// Bandrundlauf-Controller
// Kontrolliert den Bandrundlauf, ist eigentlich der Hauptbaustein(deshalb wird direkt auf PLC-Variablen zugegriffen(ohne Schnittstellenübergabe)
FUNCTION_BLOCK FB_ConvSys
VAR
    vsFB_ConvPurple : FB_Conveyor;
    vsFB_ConvOrange : FB_Conveyor;
    vsFB_ConvYellow : FB_Conveyor;
    vsFB_ConvBlue : FB_Conveyor;

    vsFB_CounterR : CTU := (PV := 0);
	vsFB_CounterL : FB_MyUpCounter;

    // Enumeration for state machine, conveyor
    eStateConveyor : E_StateConveyor;

    fbChrono : FB_Chrono;
    fbConvLapTimeStatistic : FB_ConvStatistic;
	// Maximale Rundenzeit der 10 letzten Umläufe
	tMaxLapTime: TIME;
END_VAR

// Conveyor state machine
CASE eStateConveyor OF
    E_StateConveyor.C_INIT:
        GVL_SimitSp.Qx_MotorAcwPurple := FALSE;
        GVL_SimitSp.Qx_MotorCwPurple := FALSE;
        GVL_SimitSp.Qx_FullSpeedPurple := FALSE;
        GVL_SimitSp.Qx_MotorAcwOrange := FALSE;
        GVL_SimitSp.Qx_MotorCwOrange := FALSE;
        GVL_SimitSp.Qx_FullSpeedOrange := FALSE;
        GVL_SimitSp.Qx_MotorAcwYellow := FALSE;
        GVL_SimitSp.Qx_MotorCwYellow := FALSE;
        GVL_SimitSp.Qx_FullSpeedYellow := FALSE;
        GVL_SimitSp.Qx_MotorAcwBlue := FALSE;
        GVL_SimitSp.Qx_MotorCwBlue := FALSE;
        GVL_SimitSp.Qx_FullSpeedBlue := FALSE;
        eStateConveyor := E_StateConveyor.C_NORMAL;

    E_StateConveyor.C_NORMAL:
        vsFB_ConvPurple.vix_Left := GVL_SimitSp.Ix_Left;
        vsFB_ConvPurple.vix_Right := GVL_SimitSp.Ix_Right;
        vsFB_ConvOrange.vix_Left := GVL_SimitSp.Ix_Left;
        vsFB_ConvOrange.vix_Right := GVL_SimitSp.Ix_Right;
        vsFB_ConvYellow.vix_Left := GVL_SimitSp.Ix_Left;
        vsFB_ConvYellow.vix_Right := GVL_SimitSp.Ix_Right;
        vsFB_ConvBlue.vix_Left := GVL_SimitSp.Ix_Left;
        vsFB_ConvBlue.vix_Right := GVL_SimitSp.Ix_Right;

        IF GVL_SimitSp.Ix_Enable THEN
            GVL_SimitSp.Qx_LightGreen := TRUE;
            eStateConveyor := E_StateConveyor.C_INIT_PROCESS;
        END_IF

    E_StateConveyor.C_INIT_PROCESS:
        vsFB_ConvPurple.vix_Left := FALSE;
        vsFB_ConvPurple.vix_Right := TRUE;
        vsFB_ConvOrange.vix_Left := FALSE;
        vsFB_ConvOrange.vix_Right := TRUE;
        vsFB_ConvYellow.vix_Left := FALSE;
        vsFB_ConvYellow.vix_Right := TRUE;
        vsFB_ConvBlue.vix_Left := FALSE;
        vsFB_ConvBlue.vix_Right := TRUE;

        eStateConveyor := E_StateConveyor.C_PURPLE_BACK;

    E_StateConveyor.C_PURPLE_BACK:
        IF GVL_SimitSp.Ix_RSensorPurple THEN
            vsFB_ConvPurple.vix_Left := TRUE;
            vsFB_ConvPurple.vix_Right := FALSE;

            eStateConveyor := E_StateConveyor.C_PURPLE_FORWARD;
        END_IF

    E_StateConveyor.C_PURPLE_FORWARD:
        IF GVL_SimitSp.Ix_LSensorPurple THEN
            vsFB_ConvPurple.vix_Left := FALSE;
            vsFB_ConvPurple.vix_Right := TRUE;

            eStateConveyor := E_StateConveyor.C_ORANGE_BACK;
        END_IF

    E_StateConveyor.C_ORANGE_BACK:
        IF GVL_SimitSp.Ix_RSensorOrange THEN
            vsFB_ConvOrange.vix_Left := TRUE;
            vsFB_ConvOrange.vix_Right := FALSE;

            eStateConveyor := E_StateConveyor.C_ORANGE_FORWARD;
        END_IF

    E_StateConveyor.C_ORANGE_FORWARD:
        IF GVL_SimitSp.Ix_LSensorOrange THEN
            vsFB_Convorange.vix_Left := FALSE;
            vsFB_Convorange.vix_Right := TRUE;

            eStateConveyor := E_StateConveyor.C_YELLOW_BACK;
        END_IF

    E_StateConveyor.C_YELLOW_BACK:
        IF GVL_SimitSp.Ix_RSensorYellow THEN
            vsFB_ConvYellow.vix_Left := TRUE;
            vsFB_ConvYellow.vix_Right := FALSE;

            eStateConveyor := E_StateConveyor.C_YELLOW_FORWARD;
        END_IF

    E_StateConveyor.C_YELLOW_FORWARD:
        IF GVL_SimitSp.Ix_LSensorYellow THEN
            vsFB_Convyellow.vix_Left := FALSE;
            vsFB_Convyellow.vix_Right := TRUE;

            eStateConveyor := E_StateConveyor.C_BLUE_BACK;
        END_IF

    E_StateConveyor.C_BLUE_BACK:
        IF GVL_SimitSp.Ix_RSensorBlue THEN
            vsFB_ConvBlue.vix_Left := TRUE;
            vsFB_ConvBlue.vix_Right := FALSE;

            eStateConveyor := E_StateConveyor.C_BLUE_FORWARD;
        END_IF

    E_StateConveyor.C_BLUE_FORWARD:
        IF GVL_SimitSp.Ix_LSensorblue THEN
            vsFB_Convblue.vix_Left := FALSE;
            vsFB_Convblue.vix_Right := TRUE;

            eStateConveyor := E_StateConveyor.C_PURPLE_BACK;
        END_IF

    ELSE
        eStateConveyor := E_StateConveyor.C_INIT;
END_CASE

// Reset conveyor state machine
IF GVL_SimitSp.Ix_Reset THEN
    eStateConveyor := E_StateConveyor.C_INIT;
END_IF

(*Multiinstanzaufruf von Band lila*)
vsFB_ConvPurple(vix_Power := GVL_SimitSp.Ix_PowerOn,
                vix_On := GVL_SimitSp.Ix_On,
                vix_Off := GVL_SimitSp.Ix_Off,
                vix_ManAuto := GVL_SimitSp.Ix_ManAuto,
                viw_Speed := GVL_SimitSp.Iw_SliderValue,
                vqx_MotorCw => GVL_SimitSp.Qx_MotorCwPurple,
                vqx_MotorAcw => GVL_SimitSp.Qx_MotorAcwPurple,
                vqx_VarSpeed => GVL_SimitSp.Qx_EnableVarSpeedPurple,
                vqw_Speed => GVL_SimitSp.Qw_VarSpeedPurple);
     
(*Multiinstanzaufruf von Band orange*)
vsFB_ConvOrange(vix_Power := GVL_SimitSp.Ix_PowerOn,
                vix_On := GVL_SimitSp.Ix_On,
                vix_Off := GVL_SimitSp.Ix_Off,
                vix_ManAuto := GVL_SimitSp.Ix_ManAuto,
                viw_Speed := GVL_SimitSp.Iw_SliderValue,
                vqx_MotorCw => GVL_SimitSp.Qx_MotorCwOrange,
                vqx_MotorAcw => GVL_SimitSp.Qx_MotorAcwOrange,
                vqx_VarSpeed => GVL_SimitSp.Qx_EnableVarSpeedOrange,
                vqw_Speed => GVL_SimitSp.Qw_VarSpeedOrange);

(*Multiinstanzaufruf von Band yellow*)
vsFB_ConvYellow(vix_Power := GVL_SimitSp.Ix_PowerOn,
                vix_On := GVL_SimitSp.Ix_On,
                vix_Off := GVL_SimitSp.Ix_Off,
                vix_ManAuto := GVL_SimitSp.Ix_ManAuto,
                viw_Speed := GVL_SimitSp.Iw_SliderValue,
                vqx_MotorCw => GVL_SimitSp.Qx_MotorCwYellow,
                vqx_MotorAcw => GVL_SimitSp.Qx_MotorAcwYellow,
                vqx_VarSpeed => GVL_SimitSp.Qx_EnableVarSpeedYellow,
                vqw_Speed => GVL_SimitSp.Qw_VarSpeedYellow);

(*Multiinstanzaufruf von Band blue*)
vsFB_ConvBlue(vix_Power := GVL_SimitSp.Ix_PowerOn,
                vix_On := GVL_SimitSp.Ix_On,
                vix_Off := GVL_SimitSp.Ix_Off,
                vix_ManAuto := GVL_SimitSp.Ix_ManAuto,
                viw_Speed := GVL_SimitSp.Iw_SliderValue,
                vqx_MotorCw => GVL_SimitSp.Qx_MotorCwBlue,
                vqx_MotorAcw => GVL_SimitSp.Qx_MotorAcwBlue,
                vqx_VarSpeed => GVL_SimitSp.Qx_EnableVarSpeedBlue,
                vqw_Speed => GVL_SimitSp.Qw_VarSpeedBlue);

(*Rundlauf Anzeigen*)
GVL_SimitSp.Qx_LightBlue := GVL_SimitSp.Qx_MotorAcwBlue;  (*Gegenuhrzeigersinn Kontrolleuchte*)
GVL_SimitSp.Qx_LightYellow := GVL_SimitSp.Qx_MotorCwBlue; (*Uhrzeigersinn Kontrolleuchte*)
GVL_SimitSp.Qw_Display := GVL_SimitSp.Qw_VarSpeedPurple;  (*aktuelle variable Geschwindigkeit*)

(*Eilgang auf Enable Taster*)
GVL_SimitSp.Qx_FullSpeedPurple := GVL_SimitSp.Ix_Enable;
GVL_SimitSp.Qx_FullSpeedOrange := GVL_SimitSp.Ix_Enable;
GVL_SimitSp.Qx_FullSpeedYellow := GVL_SimitSp.Ix_Enable;
GVL_SimitSp.Qx_FullSpeedBlue := GVL_SimitSp.Ix_Enable; 

// Conveyor circulation counter right
vsFB_CounterR(CU := GVL_SimitSp.Ix_RSensorPurple AND GVL_SimitSp.Qx_MotorAcwPurple);
GVL_SimitSp.Qb_74 := WORD_TO_BYTE(vsFB_CounterR.CV);

// Conveyor circulation counter left
vsFB_CounterL(CU := GVL_SimitSp.Ix_LSensorPurple AND GVL_SimitSp.Qx_MotorCwPurple);
GVL_SimitSp.Qb_75 := INT_TO_BYTE(vsFB_CounterL.CV);

// Lap time
fbChrono(bLap := GVL_SimitSp.Ix_LSensorPurple);

// Lap time history buffer
fbConvLapTimeStatistic(tLapTime := fbChrono.stLapDuration);
IF GVL_SimitSp.Ix_LSensorPurple THEN
    fbConvLapTimeStatistic.bAddValue := TRUE;
    tMaxLapTime := FC_GetMaxLapTime(fbConvLapTimeStatistic.aLapTimes);
ELSE
    fbConvLapTimeStatistic.bAddValue := FALSE;
END_IF

// Blink LED on sensor left of each conveyor
GVL_CouplerOnDesk.bSelectorSwitchLed := GVL_SimitSp.Ix_LSensorPurple OR GVL_SimitSp.Ix_LSensorBlue OR GVL_SimitSp.Ix_LSensorYellow OR GVL_SimitSp.Ix_LSensorOrange;

END_FUNCTION_BLOCK

(* stored: Version 1.1.0.1
   POU FB_ConvSys: Id {8235fbcc-99f3-4e93-85a5-6d95fab18df5}, SpecialFunc None *)
